INTERFACE ITFGesimuleerdDO

PROPERTY SensorWaarde : bool
GET
END_GET
SET
END_SET
END_PROPERTY

END_INTERFACE

(* stored: Version 1.1.0.1
   Itf ITFGesimuleerdDO: Id {76f5503f-9eb3-4de4-b711-fb6ba2555fa9}
   Property SensorWaarde: Id {48f8098c-ed33-4337-a57e-4a4066595a73}
   Get Get: Id {409eb0b4-5e73-4532-863b-3fed06b87e36}
   Set Set: Id {89ab93ab-14df-4284-9c7e-04f6524cc224} *)
